FUNCTION F_LogBuilder : I_LogBuilder
VAR_INPUT
	eLogLevel		: E_LogLevel;
	sMessages		: T_MaxString;
END_VAR

END_FUNCTION

(* stored: Version 1.1.0.1, ProductVersion 3.1.4026.8
   POU F_LogBuilder: Id {c970aefe-3199-4c53-b630-5acb322a775a}, SpecialFunc None *)
